DATA_BLOCK "OP10_GeneralAnalogDB"
VAR
  aDev : Array[1..2] of "ST_GeneralAnalog";
END_VAR
BEGIN
END_DATA_BLOCK
